FUNCTION_BLOCK EnableBehaviour IMPLEMENTS I_Task
VAR
	mcPower : Tc2_MC2.MC_Power;
	AxisReference : REFERENCE TO Tc2_MC2.AXIS_REF;
	EnableAxis : BOOL;
	State: INT;
	_Done: BOOL;
	_Error: BOOL;
	_Busy: BOOL;
END_VAR

{analysis -2}

METHOD Abort : BOOL
mcPower.Enable := mcPower.Enable_Negative := mcPower.Enable_Positive := FALSE;
_Busy := FALSE;
EnableAxis := FALSE;
Abort := TRUE;
State := 0;
END_METHOD

PROPERTY Busy : BOOL
GET
Busy := _busy;
END_GET
END_PROPERTY

METHOD Cycle : HRESULT
VAR_INPUT
END_VAR
Cycle := S_OK;
CASE State OF
	0:
		IF EnableAxis THEN
			Cycle := S_PENDING;
			_Done := FALSE;
			_Error := FALSE;
			_Busy := TRUE;
			mcPower.Enable := mcPower.Enable_Negative := mcPower.Enable_Positive := TRUE;
			mcPower.Override := 100;
			State := 10;
		END_IF
	
	10:
		IF mcPower.Status THEN
			_Busy := FALSE;
			_Done := TRUE;
			State := 20;
			Cycle := S_OK;
		END_IF
	
	20:
		IF NOT EnableAxis THEN
			_Done := FALSE;
			_Busy := TRUE;
			mcPower.Enable := mcPower.Enable_Negative := mcPower.Enable_Positive := FALSE;
			State := 30;
			Cycle := S_PENDING;
		END_IF
	30:
		IF NOT mcPower.Status THEN
			_Busy := FALSE;
			_Done := TRUE;
			State := 0;
			Cycle := S_OK;
		END_IF
	ELSE
		Cycle := E_FAIL;
END_CASE

mcPower(Axis := AxisReference);
END_METHOD

METHOD Disable : HRESULT
VAR_INPUT
	Task : REFERENCE TO I_Task;
END_VAR
IF NOT EnableAxis THEN
	Disable := S_FALSE;
ELSE
	Disable := S_OK;
	Task := THIS^;
	EnableAxis := FALSE;
END_IF
END_METHOD

PROPERTY Done : BOOL
GET
Done := _Done;
END_GET
END_PROPERTY

METHOD Enable : HRESULT
VAR_INPUT
	Task : REFERENCE TO I_Task;
END_VAR
IF EnableAxis THEN
	Enable := -1;
ELSE
	Task := THIS^;
	EnableAxis := TRUE;
	Enable := 1;
END_IF
END_METHOD

PROPERTY Error : BOOL
GET
Error := _Error;
END_GET
END_PROPERTY

METHOD FB_init : BOOL
VAR_INPUT
	bInitRetains : BOOL; // if TRUE, the retain variables are initialized (warm start / cold start)
	bInCopyCode : BOOL;  // if TRUE, the instance afterwards gets moved into the copy code (online change)
	axis : reference TO AXIS_REF;
END_VAR
AxisReference REF= axis;
END_METHOD

END_FUNCTION_BLOCK

(* stored: Version 1.1.0.1
   POU EnableBehaviour: Id {9020922a-7816-4155-9202-ac5854f794ea}, SpecialFunc None
   Method Abort: Id {93bd9e75-34cf-4a99-8cdf-c273723a870d}
   Property Busy: Id {c798d0d0-97d0-4d53-b519-da00d5dccc4f}
   Get Get: Id {c431141b-efc9-4560-8025-c7c0a08af50a}
   Method Cycle: Id {c1cf1940-bcdc-4ac4-844e-317c1f14fe0e}
   Method Disable: Id {0a54e8c6-7456-4747-8eeb-b97b9078e709}
   Property Done: Id {006aa190-9c68-4a73-bf0c-8a7f7aaf57ff}
   Get Get: Id {3155aba1-6f22-460f-ac4b-c62ed8476ecf}
   Method Enable: Id {afe5d65c-4532-4d19-b244-08cfed3445ed}
   Property Error: Id {518ce1d0-c80e-419e-af03-bf594c64bec9}
   Get Get: Id {f9e74dcb-6dbd-485e-b208-5c6b8f34d064}
   Method FB_init: Id {03d72923-bd2d-4684-847b-d6b404bc945a} *)
